// TIA Portal V18 export
DATA_BLOCK "WeatherComp"   // DB1018
{ S7_Optimized_Access := 'FALSE' }
VERSION : 0.1
// stored: AutoNumber false, DBAccessibleFromOPCUA true, IsOnlyStoredInLoadMemory false, IsWriteProtectedInAS false
   VAR
      WeatherComp { S7_SetPoint := 'True'} : "UDT_WeatherCompCurve";
   END_VAR
BEGIN
END_DATA_BLOCK
